// SIMATIC S7-200 SMART project (STEP 7-Micro/WIN SMART), CPU ST40

ORGANIZATION_BLOCK MAIN:OB1
TITLE=中断例程注释
BEGIN
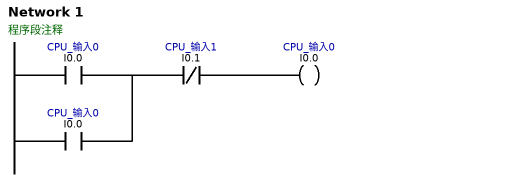
Network 1
// 程序段注释
LD     CPU_输入0:I0.0
O      CPU_输入0:I0.0
AN     CPU_输入1:I0.1
=      CPU_输入0:I0.0
Network 11
// 程序段注释
END_ORGANIZATION_BLOCK

INTERRUPT_BLOCK INT_0:INT0
TITLE=中断例程注释
BEGIN
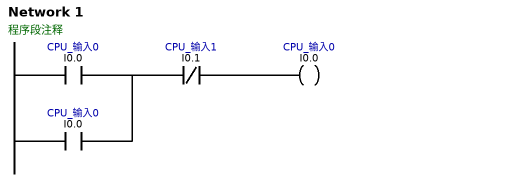
Network 1
// 程序段注释
LD     CPU_输入0:I0.0
O      CPU_输入0:I0.0
AN     CPU_输入1:I0.1
=      CPU_输入0:I0.0
END_INTERRUPT_BLOCK
